// TIA Portal V21 export
VAR_GLOBAL   // PLC tag table "默认变量表"
   报文750当前扭矩 AT %IW92 : Int;
   报文750附加扭矩给定 AT %QW88 : Int;
   报文750上限扭矩限定 AT %QW90 : Int;
   报文750下限扭矩限定 AT %QW92 : Int;
   System_Byte AT %MB8190 : Byte;
   FirstScan AT %M8190.0 : Bool;
   DiagStatusUpdate AT %M8190.1 : Bool;
   AlwaysTRUE AT %M8190.2 : Bool;
   AlwaysFALSE AT %M8190.3 : Bool;
   Clock_Byte AT %MB8191 : Byte;
   Clock_10Hz AT %M8191.0 : Bool;
   Clock_5Hz AT %M8191.1 : Bool;
   "Clock_2.5Hz" AT %M8191.2 : Bool;
   Clock_2Hz AT %M8191.3 : Bool;
   "Clock_1.25Hz" AT %M8191.4 : Bool;
   Clock_1Hz AT %M8191.5 : Bool;
   "Clock_0.625Hz" AT %M8191.6 : Bool;
   "Clock_0.5Hz" AT %M8191.7 : Bool;
   TRIG_P1 AT %M0.4 : Bool;
   JogModePuse AT %M0.6 : Bool;
   PosModePuse AT %M0.7 : Bool;
   HomeModePuse AT %M1.0 : Bool;
   TRIG_P2 AT %M0.5 : Bool;
END_VAR
